{attribute 'qualified_only'}
{attribute 'strict'}
TYPE ENUM_MotionRequest :
(
	WAIT := 0,
	INTERRUPT := 1,
	ABORT := 2
);
END_TYPE

(* stored: Version 1.1.0.1, ProductVersion 3.1.4022.18
   DUT ENUM_MotionRequest: Id {0497ccec-2aee-4f07-877c-128fdd95a4b7} *)
